FUNCTION_BLOCK FB_EPSSamplePaddleGasNeedle IMPLEMENTS I_EPSSamplePaddleGasNeedle
VAR
    fbEPSSamplePaddleForwardZ : FB_EPS;
    fbEPSSamplePaddleBackwardZ : FB_EPS;

    fbEPSGasNeedleForwardZ : FB_EPS;
    fbEPSGasNeedleBackwardZ : FB_EPS;

    fSamplePaddleZOut : LREAL := 100.0; // Greater than this number is out
    fGasNeedleZOut : LREAL := 85.0; // Less than this number is out
END_VAR


METHOD PRIVATE AllowGasNeedleZToMoveIn

fbEPSGasNeedleForwardZ.setBit(nBits := 0, bValue := TRUE);
fbEPSGasNeedleForwardZ.setMessage(message := 'EPS is permitting forward motion.');
END_METHOD


METHOD PRIVATE AllowSamplePaddleZToMoveIn

fbEPSSamplePaddleBackwardZ.setBit(nBits := 0, bValue := TRUE);
fbEPSSamplePaddleBackwardZ.setMessage(message := 'EPS is permitting backward motion.');
END_METHOD


METHOD CheckAndActivateIfRequired
VAR_IN_OUT
    StageZSamplePaddle	: lcls_twincat_motion.ST_MotionStage;
    StageZGasNeedle	: lcls_twincat_motion.ST_MotionStage;
END_VAR

// Sample Paddle
fbEPSSamplePaddleForwardZ(eps := StageZSamplePaddle.stEPSForwardEnable);
fbEPSSamplePaddleForwardZ.setDescription(desciption := 'Sample Paddle Stage Z Forward EPS');

fbEPSSamplePaddleBackwardZ(eps := StageZSamplePaddle.stEPSBackwardEnable);
fbEPSSamplePaddleBackwardZ.setDescription(desciption := 'Sample Paddle Stage Z Backward EPS');

IF GasNeedleZIsOut(StageZGasNeedle := StageZGasNeedle) THEN
    AllowSamplePaddleZToMoveIn();
ELSE
    PreventSamplePaddleZFromMovingIn();
    StageZSamplePaddle.sCustomErrorMessage := 'Cannot move any further in because Gas Needle Z is in.';
END_IF

// Gas Needle
fbEPSGasNeedleForwardZ(eps := StageZGasNeedle.stEPSForwardEnable);
fbEPSGasNeedleForwardZ.setDescription(desciption := 'Gas Needle Stage Z Forward EPS');

IF SamplePaddleZIsOut(StageZSamplePaddle := StageZSamplePaddle) THEN
    AllowGasNeedleZToMoveIn();
ELSE
    PreventGasNeedleZFromMovingIn();
    StageZGasNeedle.sCustomErrorMessage := 'Cannot move any further in because Sample Paddle Z is in.';
END_IF

fbEPSGasNeedleBackwardZ(eps := StageZGasNeedle.stEPSBackwardEnable);
fbEPSGasNeedleBackwardZ.setDescription(desciption := 'Gas Needle Stage Z Backward EPS');
END_METHOD


METHOD PRIVATE GasNeedleZIsOut : BOOL
VAR_INPUT
    StageZGasNeedle	: lcls_twincat_motion.ST_MotionStage;
END_VAR

GasNeedleZIsOut := StageZGasNeedle.Axis.NcToPlc.ActPos <= fGasNeedleZOut;
END_METHOD


METHOD PRIVATE PreventGasNeedleZFromMovingIn

fbEPSGasNeedleForwardZ.setBit(nBits := 0, bValue := FALSE);
fbEPSGasNeedleForwardZ.setMessage(message := 'Cannot move in when Sample Paddle Z is not out.');
END_METHOD


METHOD PRIVATE PreventSamplePaddleZFromMovingIn

fbEPSSamplePaddleBackwardZ.setBit(nBits := 0, bValue := FALSE);
fbEPSSamplePaddleBackwardZ.setMessage(message := 'Cannot move in when Gas Needle Z is not out.');
END_METHOD


METHOD PRIVATE SamplePaddleZIsOut : BOOL
VAR_INPUT
    StageZSamplePaddle	: lcls_twincat_motion.ST_MotionStage;
END_VAR

SamplePaddleZIsOut := StageZSamplePaddle.Axis.NcToPlc.ActPos >= fSamplePaddleZOut;
END_METHOD

END_FUNCTION_BLOCK

(* stored: Version 1.1.0.1, ProductVersion 3.1.4022.18
   POU FB_EPSSamplePaddleGasNeedle: Id {2e0cf1df-b00b-4bd4-b07c-167344109ad0}, SpecialFunc None
   Method AllowGasNeedleZToMoveIn: Id {aea5ef35-815f-4db6-9bd5-85f20ecb5f31}
   Method AllowSamplePaddleZToMoveIn: Id {df323478-dad5-4e44-ac80-db0ff4f4c6bc}
   Method CheckAndActivateIfRequired: Id {daed7d29-9c62-4a7b-a62b-88629e881b75}
   Method GasNeedleZIsOut: Id {e47d70b8-9a9d-4b55-9c9a-a5bc868700cd}
   Method PreventGasNeedleZFromMovingIn: Id {a702c8da-f7fe-47c9-9879-886e32025bfd}
   Method PreventSamplePaddleZFromMovingIn: Id {1083b9a6-3c04-46ec-bc72-bcfd74bf3154}
   Method SamplePaddleZIsOut: Id {28504932-4cc0-4aa9-8e94-e0ee04d036be} *)
